TYPE ST_CyclicMessageDetection :
STRUCT
  ev: EventMessage;
  message_submitted: BOOL;
END_STRUCT
END_TYPE

(* stored: Version 1.1.0.1, ProductVersion 3.1.4024.9
   DUT ST_CyclicMessageDetection: Id {691dc274-62d5-43ab-98ac-3f694b7348db} *)
